Fanuc KAREL source: kb00163.KL

-- PROVISIONAL review KL for V940-1; original PC SHA256 96c6678442d074cde84bde892a319c1da9b81d542d13f475802f541c269a9fac
-- Incomplete behavior may be omitted. Consult companion uncertainty JSON. Do not deploy.
PROGRAM KB00163
%NOLOCKGROUP
BEGIN
  -- V9_ZERO_TABLE_METADATA_HINT layout=0002_ascii; no indexed target words; source/name/runtime held
  -- UNRESOLVED_PC offsets 5-12; opcodes 9D,23
  -- UNRESOLVED_PC offsets 17-35; opcodes 27,22,22,27,9D,31
  -- UNRESOLVED_PC offsets 40-44; opcodes 7F
END KB00163
